// TwinCAT 3 PLC project BPC_PPA
// ProgramVersion: 3.1.4024.0
// libraries:
//   Tc2_Standard, * (Beckhoff Automation GmbH)
//   Tc2_System, * (Beckhoff Automation GmbH)
//   Tc3_Module, * (Beckhoff Automation GmbH)
//   VisuSymbols,3.5.10.0,System
// project tree:
//   / GlobalTextList.TcGTLO, PlcTask.TcTTO, Visualization Manager.TcVMO (not stored)
//   GVLs/ GVL.TcGVL, IO.TcGVL
//   POUs/ IOmap.TcPOU, MAIN.TcPOU, P_regulator.TcPOU
//   VISUs/ Visualization.TcVIS
// real-time tasks:
//   TASK PlcTask: cycle T#10ms, priority 20, ADS port 350

CONFIGURATION BPC_PPA
    RESOURCE PLC ON TwinCAT3
        TASK PlcTask(INTERVAL := T#10ms, PRIORITY := 20);
        PROGRAM MAIN WITH PlcTask : MAIN;
    END_RESOURCE
END_CONFIGURATION

// ---- GVLs/GVL.TcGVL
VAR_GLOBAL
    mb_Input_Coils : ARRAY [0..20] OF BOOL;
    mb_Output_Coils : ARRAY [0..20] OF BOOL;
    mb_Input_Registers : ARRAY [0..20] OF WORD;
    mb_Output_Registers : ARRAY [0..20] OF WORD;
END_VAR

// ---- GVLs/IO.TcGVL
{attribute 'qualified_only'}
VAR_GLOBAL
	// Analog Inputs
	StorageSupportPosition	: WORD;	// Pozice supportu skladovacího manipulátoru [0..27648]
	StorageCarriagePosition	: WORD;	// Pozice vozíku skladovacího manipulátoru [0..27648]
	
	// Digital Inputs
	SensorBoxStart			: BOOL;	// Sensor přítomnosti bedny na vstupu velkého dopravníkového pásu [0/1]
	SensorBoxHandling		: BOOL;	// Sensor přítomnosti bedny v pracovním prostoru překládacího manipulátoru [0/1]
	SensorBoxHandled		: BOOL;	// Sensor přítomnosti bedny na konci velkého dopravníkového pásu [0/1]
	SensorBoxStoring		: BOOL;	// Sensor přítomnosti bedny na naskladňovací pozici zakládacího dopravníku [0/1]
	SensorCanNew			: BOOL;	// Sensor přítomnosti nové plechovky na malém dopravníkovém pásu [0/1]
	SensorCanPrepare		: BOOL;	// Sensor přítomnosti plechovky uprostřed malého dopravníkového pásu [0/1]
	SensorCanHandling		: BOOL;	// Sensor přítomnosti plechovky v pracovním prostoru překládacího manipulátoru [0/1]
	ConvCanMoving			: BOOL;	// Signalizace pohybu motoru malého dopravníkového pásu [0/1]
	ConvBoxMoving			: BOOL;	// Signalizace pohybu motoru velkého dopravníkového pásu [0/1]
	ConvLoadMoving			: BOOL;	// Signalizace pohybu motoru zakládacího dopravníkového pásu [0/1]
	StorageSupportMoving	: BOOL;	// Signalizace pohybu motoru supportu skladovacího manipulátoru [0/1]
	StorageCarriageMoving	: BOOL;	// Signalizace pohybu motoru vozíku skladovacího manipulátoru [0/1]
	RoboticArmMoving		: BOOL;	// Signalizace vykonávání programového cyklu 6-osého robotického manipulátoru [0/1]
	HandlingMoving			: BOOL;	// Signalizace vykonávání programového cyklu překládacího manipulátoru [0/1]

	// Analog Outputs
	RoboticArmProgram		: WORD;	// Číslo programu pro vykonání 6-osým manipulátorem [0 .. základní pozice, 1 ..uchopení bedny, 2 .. položení bedny na pás]
	HandlingProgram			: WORD;	// Číslo programu pro vykonání překládacím manipulátorem [0 .. základní pozice, 1 .. přenesení na první pozici, 2 .. přenesení na druhou pozici, 3 .. přenesení na třetí pozici]
	ConvCanSpeed			: WORD;	// Rychlost motoru malého dopravníku [0..27648]
	ConvBoxSpeed			: WORD;	// Rychlost motoru velkého dopravníku [0..27648]
	ConvLoadSpeed			: WORD;	// Rychlost motoru zakládacího dopravníku [0..27648]
	StorageSupportSpeed		: WORD;	// Rychlost motoru supportu skladovacího manipulátoru [0..27648]
	StorageCarriageSpeed	: WORD;	// Rychlost motoru vozíku skladovacího manipulátoru [0..27648]
	
	// Digital Outputs
	RoboticArmStartCycle	: BOOL;	// Start programového cyklu 6-osého manipulátoru [náběžná hrana]
	HandlingStartCycle		: BOOL;	// Start programového cyklu překládacího manipulátoru [náběžná hrana]
	StorageLoad				: BOOL;	// Aktivace válce (ventilu) plošiny skladovacího manipulátoru DO naskladňovací polohy [0/1]
	StorageUnload			: BOOL;	// Aktivace válce (ventilu) plošiny skladovacího manipulátoru provyskladňovací polohy [0/1]
	ConvCanEnable			: BOOL;	// Povolení frekvenčního měniče motoru malého dopravníku [0/1]
	ConvCanForward			: BOOL;	// Aktivace chodu motoru malého dopravníku standardním směrem [0/1]
	ConvCanBackward			: BOOL;	// Aktivace chodu motoru malého dopravníku zpětným směrem [0/1]
	ConvBoxEnable			: BOOL;	// Povolení frekvenčního měniče motoru velkého dopravníku [0/1]
	ConvBoxForward			: BOOL;	// Aktivace chodu motoru velkého dopravníku standardním směrem [0/1]
	ConvBoxBackward			: BOOL;	// Aktivace chodu motoru velkého dopravníku zpětným směrem [0/1]
	ConvLoadEnable			: BOOL;	// Povolení frekvenčního měniče motoru zakládacího dopravníku [0/1]
	ConvLoadForward			: BOOL;	// Aktivace chodu motoru zakládacího dopravníku standardním směrem [0/1]
	ConvLoadBackward		: BOOL;	// Aktivace chodu motoru zakládacího dopravníku zpětným směrem [0/1]
	StorageSupportEnable	: BOOL;	// Povolení frekvenčního měniče motoru supportu skladovacího manipulátoru [0/1]
	StorageSupportForward	: BOOL;	// Aktivace chodu motoru supportu skladovacího manipulátoru standardním směrem [0/1]
	StorageSupportBackward	: BOOL;	// Aktivace chodu motoru supportu skladovacího manipulátoru zpětným směrem [0/1]
	StorageCarriageEnable	: BOOL;	// Povolení frekvenčního měniče motoru vozíku skladovacího manipuátoru [0/1]
	StorageCarriageForward	: BOOL;	// Aktivace chodu motoru vozíku skladovacího manipulátoru standardním směrem [0/1]
	StorageCarriageBackward	: BOOL;	// Aktivace chodu motoru vozíku skladovacího manipulátoru zpětným směrem [0/1]	
END_VAR

// ---- POUs/MAIN.TcPOU
PROGRAM MAIN
VAR CONSTANT
	//hlavni stavovy automat
	WAITING_FOR_START : USINT := 0;
	INIT_ROBOTS : USINT := 1; //inicializace handleru plechovek i velkeho robota
	INIT_ROBOTS_WAIT : USINT := 2; //cekaci stav, protoze pouzivam casovac
	GRAB_BOX : USINT := 3;
	GRAB_BOX_WAIT : USINT := 4;
	PUT_BOX : USINT := 5;
	PUT_BOX_WAIT : USINT := 6;
	DRIVE_BOX_TO_HANDLER : USINT := 7;
	HANDLE_CAN1 : USINT := 8;
	HANDLE_CAN1_WAIT : USINT := 9;
	HANDLE_CAN2 : USINT := 10;
	HANDLE_CAN2_WAIT : USINT := 11;
	HANDLE_CAN3 : USINT := 12;
	HANDLE_CAN3_WAIT : USINT := 13;
	CANS_HANDLED : USINT := 14;
	STORAGE_INIT : USINT := 15;
	STORAGE_INIT_WAIT : USINT := 16;
	GET_BOX_STORE : USINT := 17;
	GET_BOX_STORE_WAIT : USINT := 18;
	STORAGE_HANDLER_TO_BOX : USINT := 19;
	STORAGE_HANDLER_TO_BOX_WAIT: USINT := 20;
	LOAD_BOX : USINT := 21;
	LOAD_BOX_WAIT : USINT := 22;
	DRIVE_BOX_TO_STORE : USINT := 23;
	DRIVE_BOX_TO_STORE_WAIT : USINT := 24;
	BOX_UNLOAD : USINT := 25;
	BOX_UNLOAD_WAIT : USINT := 26;
	LAY_BOX : USINT := 27;
	STORING_DONE : USINT := 28;
END_VAR

VAR
	MainState : USINT := WAITING_FOR_START;
	StartProcess : BOOL := FALSE;
	CanSpeed : WORD := 1900;
	ConvSpeed : WORD := 2800;
	BoxAtTheEnd : BOOL := FALSE;
	TON_DelayCycle : TON;
	x : ARRAY [0..10] OF WORD := [25580, 23000, 20420, 17845, 15260, 12700, 10120, 7520, 4940, 2380, 750];
	y : ARRAY [0..5] OF WORD := [23750, 19142, 14535, 9927, 5318, 710];
	//FirstBoxDriven : BOOL := FALSE;
	BoxesStored : USINT := 0;
	ID : ARRAY [0..5] OF USINT := [2,5,6,3,9,4];
	P_RegulatorX : P_regulator;
	P_RegulatorY : P_regulator;
	yPosition : WORD := 0;
	xPosition : WORD := 0;
	RoboticArmStart : BOOL := FALSE;
	CentralStop : BOOL := FALSE;
END_VAR


IOmap(); //namapuj vstupy a vystupy
IF CentralStop THEN
	IO.ConvBoxEnable := 0;
	IO.ConvCanEnable := 0;
	IO.StorageSupportEnable := 0;
	IO.StorageCarriageEnable := 0;
	IO.StorageSupportEnable := 0;
END_IF

CASE MainState OF
	WAITING_FOR_START:
		IF StartProcess THEN
			MainState := INIT_ROBOTS;
		END_IF
		
	INIT_ROBOTS:
		IO.HandlingProgram := IO.RoboticArmProgram := 0;
		IO.HandlingStartCycle := IO.RoboticArmStartCycle := 1;
		TON_DelayCycle(IN := TRUE, PT := T#1S);
		IF TON_DelayCycle.Q THEN
			TON_DelayCycle(IN := 0);
			IF NOT IO.RoboticArmMoving AND NOT IO.HandlingMoving THEN
				IO.HandlingStartCycle := IO.RoboticArmStartCycle := 0;
				MainState := INIT_ROBOTS_WAIT;
			END_IF
		END_IF
		
	INIT_ROBOTS_WAIT:
		TON_DelayCycle(IN := TRUE, PT := T#1S);
		IF TON_DelayCycle.Q THEN
			TON_DelayCycle(IN := 0); 
			MainState := GRAB_BOX;
		END_IF
		
	GRAB_BOX:
		IO.RoboticArmProgram := 1;
		IO.RoboticArmStartCycle := 1;
		TON_DelayCycle(IN := TRUE, PT := T#1S);
		IF TON_DelayCycle.Q THEN
			TON_DelayCycle(IN := 0);
			IF NOT IO.RoboticArmMoving THEN
				IO.RoboticArmStartCycle := 0;
				MainState := GRAB_BOX_WAIT;
			END_IF
		END_IF
		
	GRAB_BOX_WAIT:
		TON_DelayCycle(IN := TRUE, PT := T#1S);
		IF TON_DelayCycle.Q THEN
			TON_DelayCycle(IN := 0);
			MainState := PUT_BOX;
		END_IF
	
	PUT_BOX:
		IO.RoboticArmProgram := 2;
		IO.RoboticArmStartCycle := 1;
		TON_DelayCycle(IN := TRUE, PT := T#1S);
		IF TON_DelayCycle.Q THEN 
			TON_DelayCycle(IN := 0);
			IF NOT IO.RoboticArmMoving THEN
				IO.RoboticArmStartCycle := 0;
				MainState := PUT_BOX_WAIT;
			END_IF
			
		END_IF
		
	PUT_BOX_WAIT:
		TON_DelayCycle(IN := TRUE, PT := T#1S);
		IF TON_DelayCycle.Q THEN
			TON_DelayCycle(IN := 0);
			MainState := DRIVE_BOX_TO_HANDLER;
		END_IF
		
	DRIVE_BOX_TO_HANDLER:
		
		IF IO.SensorBoxHandling THEN
			IO.ConvBoxEnable := 0;
			MainState := HANDLE_CAN1;
		ELSE
			IO.ConvBoxEnable := 1;
		END_IF
		
		
	HANDLE_CAN1:
		IO.HandlingProgram := 1;
		IO.HandlingStartCycle := 1;
		TON_DelayCycle(IN := TRUE, PT := T#1S);
		IF TON_DelayCycle.Q THEN
			TON_DelayCycle(IN := 0);
			IF NOT IO.HandlingMoving THEN
				IO.HandlingStartCycle := 0; 
				MainState := HANDLE_CAN1_WAIT;
			END_IF
		END_IF
		
	HANDLE_CAN1_WAIT:
		TON_DelayCycle(IN := TRUE, PT := T#1S);
		IF TON_DelayCycle.Q THEN
			TON_DelayCycle(IN := 0); 
			MainState := HANDLE_CAN2;
		END_IF
		
	HANDLE_CAN2:
		TON_DelayCycle(IN := TRUE, PT := T#1S);
		IO.HandlingProgram := 2;
		IO.HandlingStartCycle := 1;
		IF TON_DelayCycle.Q THEN
			TON_DelayCycle(IN := 0);
			IF NOT IO.HandlingMoving THEN
				IO.HandlingStartCycle := 0;
				MainState := HANDLE_CAN2_WAIT;
			END_IF
		END_IF
		
	HANDLE_CAN2_WAIT:
		TON_DelayCycle(IN := TRUE, PT := T#1S);
		IF TON_DelayCycle.Q THEN
			TON_DelayCycle(IN := 0); 
			MainState := HANDLE_CAN3;
		END_IF
		
	HANDLE_CAN3:
		TON_DelayCycle(IN := TRUE, PT := T#1S);
		IO.HandlingProgram := 3;
		IO.HandlingStartCycle := 1;
		IF TON_DelayCycle.Q THEN
			TON_DelayCycle(IN := 0);
			IF NOT IO.HandlingMoving THEN
				IO.HandlingStartCycle := 0; 
				MainState := HANDLE_CAN3_WAIT;
			END_IF
		END_IF
		
	HANDLE_CAN3_WAIT:
		TON_DelayCycle(IN := TRUE, PT := T#1S);
		IF TON_DelayCycle.Q THEN
			TON_DelayCycle(IN := 0);
			MainState := CANS_HANDLED;
		END_IF	
	
	CANS_HANDLED:
		MainState := GET_BOX_STORE;
		IO.ConvBoxEnable := 1;
	
	STORAGE_INIT:
		TON_DelayCycle(IN := TRUE, PT := T#1S);
		
		P_RegulatorX.SetpointPos := 750;
		P_RegulatorY.SetpointPos := 1100;
		
		IF TON_DelayCycle.Q THEN
			TON_DelayCycle(IN := 0);
			IF NOT IO.StorageCarriageMoving AND NOT IO.StorageSupportMoving THEN
				
				MainState := STORAGE_INIT_WAIT;
			END_IF
		
		END_IF
		
	STORAGE_INIT_WAIT:
		TON_DelayCycle(IN := TRUE, PT := T#1S);
		IF TON_DelayCycle.Q THEN
			TON_DelayCycle(IN := 0); 
			MainState := GET_BOX_STORE;
		END_IF
		
	GET_BOX_STORE:
		IO.StorageCarriageEnable := IO.StorageSupportEnable := 1;
		IF IO.SensorBoxStoring THEN
			TON_DelayCycle(IN := TRUE, PT := T#1S);
			P_RegulatorX.SetpointPos := 750;
			P_RegulatorY.SetpointPos := 1100;	
			IF TON_DelayCycle.Q THEN
					IF NOT IO.StorageSupportMoving AND NOT IO.StorageCarriageMoving THEN
						
						MainState := GET_BOX_STORE_WAIT;
					END_IF
			END_IF
		END_IF
		
	GET_BOX_STORE_WAIT:
		TON_DelayCycle(IN := TRUE, PT := T#1S);
		IF TON_DelayCycle.Q THEN
			TON_DelayCycle(IN := 0); 
			
			MainState := STORAGE_HANDLER_TO_BOX;
		END_IF
		
	STORAGE_HANDLER_TO_BOX:
		TON_DelayCycle(IN := TRUE, PT := T#2S);
		IF TON_DelayCycle.Q THEN
			P_RegulatorY.SetpointPos := 2100;
			IO.StorageLoad := 1;
			MainState := STORAGE_HANDLER_TO_BOX_WAIT;
		END_IF
	
	STORAGE_HANDLER_TO_BOX_WAIT:
		TON_DelayCycle(IN := TRUE, PT := T#2S);
		IF TON_DelayCycle.Q THEN
			
			TON_DelayCycle(IN := FALSE);
			MainState := LOAD_BOX;
		END_IF
		
	LOAD_BOX:
		TON_DelayCycle(IN := TRUE, PT := T#2S);
		IF TON_DelayCycle.Q THEN
			TON_DelayCycle(IN := FALSE);
			IO.StorageLoad := 0;
			MainState := LOAD_BOX_WAIT;
		END_IF
		
	LOAD_BOX_WAIT:
		TON_DelayCycle(IN := TRUE, PT := T#2S);
		IF TON_DelayCycle.Q THEN
			TON_DelayCycle(IN := FALSE);
			MainState := DRIVE_BOX_TO_STORE;
		END_IF
	
		
	DRIVE_BOX_TO_STORE: 
		TON_DelayCycle(IN := TRUE, PT := T#1S);
		IF TON_DelayCycle.Q THEN
			TON_DelayCycle(IN := FALSE);
				P_RegulatorX.SetpointPos := x[ID[BoxesStored]];
				P_RegulatorY.SetpointPos := y[BoxesStored] + 400;
			MainState := DRIVE_BOX_TO_STORE_WAIT; 
		END_IF
		
	DRIVE_BOX_TO_STORE_WAIT:
		TON_DelayCycle(IN := TRUE, PT := T#1S);
		IF TON_DelayCycle.Q THEN
			TON_DelayCycle(IN := FALSE);
			MainState := BOX_UNLOAD;
		END_IF
		
	BOX_UNLOAD: 
		TON_DelayCycle(IN := TRUE, PT := T#1S);
		IF TON_DelayCycle.Q THEN
			IF NOT IO.StorageCarriageMoving AND NOT IO.StorageSupportMoving THEN
				TON_DelayCycle(IN := FALSE);
				IO.StorageUnload := 1;
				MainState := BOX_UNLOAD_WAIT;
			END_IF
		END_IF
	BOX_UNLOAD_WAIT:
		TON_DelayCycle(IN := TRUE, PT := T#1S);
		IF TON_DelayCycle.Q THEN
				TON_DelayCycle(IN := FALSE);
				MainState := LAY_BOX;
				P_RegulatorY.SetpointPos := P_RegulatorY.SetpointPos - 400;
		END_IF
		
	LAY_BOX:
		TON_DelayCycle(IN := TRUE, PT := T#1S);
		IF TON_DelayCycle.Q THEN
			IF NOT IO.StorageCarriageMoving AND NOT IO.StorageSupportMoving THEN
				TON_DelayCycle(IN := FALSE);
				IO.StorageUnload := 0;
				IF BoxesStored < 5 THEN
					MainState := GRAB_BOX;
					BoxesStored := BoxesStored + 1;
				ELSE
					MainState := STORING_DONE;
				END_IF
			END_IF 
			
		END_IF
		
END_CASE

IF IO.SensorBoxHandled THEN
	BoxAtTheEnd := TRUE;
END_IF

//maly dopravnik
IO.ConvCanSpeed := CanSpeed;
IO.ConvCanForward := TRUE;
IO.ConvCanEnable := NOT IO.SensorCanHandling AND MainState > WAITING_FOR_START;
StartProcess := FALSE;

//velky dopravnik
IO.ConvBoxSpeed := ConvSpeed;
IO.ConvBoxForward := TRUE;

//zakladaci dopravnik
IO.ConvLoadSpeed := ConvSpeed;
IO.ConvLoadForward := TRUE;
IO.ConvLoadEnable := BoxAtTheEnd AND NOT IO.SensorBoxStoring;

P_RegulatorX(CurrentPos := IO.StorageSupportPosition, DecelerationLength := 15000);
IO.StorageSupportSpeed := REAL_TO_WORD(P_RegulatorX.Speed);
IO.StorageSupportForward := P_RegulatorX.MoveForward;
IO.StorageSupportBackward := P_RegulatorX.MoveBackward;

P_RegulatorY(CurrentPos := IO.StorageCarriagePosition, DecelerationLength := 17000);
IO.StorageCarriageSpeed := REAL_TO_WORD(P_RegulatorY.Speed);
IO.StorageCarriageForward := P_RegulatorY.MoveForward;
IO.StorageCarriageBackward := P_RegulatorY.MoveBackward;

END_PROGRAM

// ---- POUs/P_regulator.TcPOU
FUNCTION_BLOCK P_regulator
VAR CONSTANT
    //FSM states
    NOT_MOVING : USINT := 0;
    MOVING : USINT := 1;

    OUTER_POS_TOL : REAL := 10;
    INNER_POS_TOL : REAL := 5;

END_VAR

VAR
    MoveState : USINT := NOT_MOVING;

    DesiredSpeed : REAL;
    DecelerationRatio : REAL;

END_VAR

VAR_INPUT
    CurrentPos : REAL;
    SetpointPos : REAL;
    MaxSpeed : REAL := 13000;
    DecelerationLength : REAL := 18000;
END_VAR

VAR_OUTPUT
    Speed : REAL;
    MoveForward : BOOL;
    MoveBackward : BOOL;
END_VAR

CASE MoveState OF
    NOT_MOVING:
        IF SetpointPos - CurrentPos > OUTER_POS_TOL THEN
            MoveForward := TRUE;
            MoveBackward := FALSE;
            MoveState := MOVING;
        ELSIF CurrentPos - SetpointPos > OUTER_POS_TOL THEN
            MoveForward := FALSE;
            MoveBackward := TRUE;
            MoveState := MOVING;
        END_IF

    MOVING:
        IF NOT (MoveForward AND SetpointPos - CurrentPos < INNER_POS_TOL OR MoveBackward AND CurrentPos - SetpointPos < INNER_POS_TOL) THEN
           IF DecelerationLength > 0 THEN
				DecelerationRatio := ABS(SetpointPos - CurrentPos) / DecelerationLength;
				IF DecelerationRatio > 1 THEN
					DecelerationRatio := 1;
				END_IF
			ELSE
				DecelerationRatio := 1;
			END_IF
            DesiredSpeed := MaxSpeed * DecelerationRatio;
        ELSE
			DesiredSpeed := 0;
            MoveForward := MoveBackward := FALSE;
            MoveState := NOT_MOVING;
			
        END_IF

END_CASE
Speed := DesiredSpeed;

END_FUNCTION_BLOCK

// ---- POUs/IOmap.TcPOU
PROGRAM IOmap
VAR
END_VAR

// Analog Inputs
IO.StorageSupportPosition 		:= GVL.mb_Output_Registers[1];		// Pozice supportu skladovacího manipulátoru [0..27648]
IO.StorageCarriagePosition 		:= GVL.mb_Output_Registers[2];		// Pozice vozíku skladovacího manipulátoru [0..27648]
	
// Digital Inputs
IO.SensorBoxStart 				:= GVL.mb_Output_Registers[0].0;	// Sensor přítomnosti bedny na vstupu velkého dopravníkového pásu [0/1]
IO.SensorBoxHandling 			:= GVL.mb_Output_Registers[0].1;	// Sensor přítomnosti bedny v pracovním prostoru překládacího manipulátoru [0/1]
IO.SensorBoxHandled 			:= GVL.mb_Output_Registers[0].2;	// Sensor přítomnosti bedny na konci velkého dopravníkového pásu [0/1]
IO.SensorBoxStoring 			:= GVL.mb_Output_Registers[0].3;	// Sensor přítomnosti bedny na naskladňovací pozici zakládacího dopravníku [0/1]
IO.SensorCanNew 				:= GVL.mb_Output_Registers[0].4;	// Sensor přítomnosti nové plechovky na malém dopravníkovém pásu [0/1]
IO.SensorCanPrepare 			:= GVL.mb_Output_Registers[0].5;	// Sensor přítomnosti plechovky uprostřed malého dopravníkového pásu [0/1]
IO.SensorCanHandling 			:= GVL.mb_Output_Registers[0].6;	// Sensor přítomnosti plechovky v pracovním prostoru překládacího manipulátoru [0/1]
IO.ConvCanMoving 				:= GVL.mb_Output_Registers[0].7;	// Signalizace pohybu motoru malého dopravníkového pásu [0/1]
IO.ConvBoxMoving 				:= GVL.mb_Output_Registers[0].8;	// Signalizace pohybu motoru velkého dopravníkového pásu [0/1]
IO.ConvLoadMoving 				:= GVL.mb_Output_Registers[0].9;	// Signalizace pohybu motoru zakládacího dopravníkového pásu [0/1]
IO.StorageSupportMoving 		:= GVL.mb_Output_Registers[0].10;	// Signalizace pohybu motoru supportu skladovacího manipulátoru [0/1]
IO.StorageCarriageMoving 		:= GVL.mb_Output_Registers[0].11;	// Signalizace pohybu motoru vozíku skladovacího manipulátoru [0/1]
IO.RoboticArmMoving 			:= GVL.mb_Output_Registers[0].12;	// Signalizace vykonávání programového cyklu 6-osého robotického manipulátoru [0/1]
IO.HandlingMoving 				:= GVL.mb_Output_Registers[0].13;	// Signalizace vykonávání programového cyklu překládacího manipulátoru [0/1]

// Analog Outputs
GVL.mb_Input_Registers[2] 		:= IO.RoboticArmProgram;			// Číslo programu pro vykonání 6-osým manipulátorem [0 .. základní pozice, 1 ..uchopení bedny, 2 .. položení bedny na pás]
GVL.mb_Input_Registers[3] 		:= IO.HandlingProgram;				// Číslo programu pro vykonání překládacím manipulátorem [0 .. základní pozice, 1 .. přenesení na první pozici, 2 .. přenesení na druhou pozici, 3 .. přenesení na třetí pozici]
GVL.mb_Input_Registers[4] 		:= IO.ConvCanSpeed;					// Rychlost motoru malého dopravníku [0..27648]
GVL.mb_Input_Registers[5] 		:= IO.ConvBoxSpeed;					// Rychlost motoru velkého dopravníku [0..27648]
GVL.mb_Input_Registers[6] 		:= IO.ConvLoadSpeed;				// Rychlost motoru zakládacího dopravníku [0..27648]
GVL.mb_Input_Registers[7] 		:= IO.StorageSupportSpeed;			// Rychlost motoru supportu skladovacího manipulátoru [0..27648]
GVL.mb_Input_Registers[8] 		:= IO.StorageCarriageSpeed;			// Rychlost motoru vozíku skladovacího manipulátoru [0..27648]

// Digital Outputs
GVL.mb_Input_Registers[0].0 	:= IO.RoboticArmStartCycle;			// Start programového cyklu 6-osého manipulátoru [náběžná hrana]
GVL.mb_Input_Registers[0].1 	:= IO.HandlingStartCycle;			// Start programového cyklu překládacího manipulátoru [náběžná hrana]
GVL.mb_Input_Registers[0].2 	:= IO.StorageLoad;					// Aktivace válce (ventilu) plošiny skladovacího manipulátoru DO naskladňovací polohy [0/1]
GVL.mb_Input_Registers[0].3 	:= IO.StorageUnload;				// Aktivace válce (ventilu) plošiny skladovacího manipulátoru provyskladňovací polohy [0/1]
GVL.mb_Input_Registers[0].4 	:= IO.ConvCanEnable;				// Povolení frekvenčního měniče motoru malého dopravníku [0/1]
GVL.mb_Input_Registers[0].5 	:= IO.ConvCanForward;				// Aktivace chodu motoru malého dopravníku standardním směrem [0/1]
GVL.mb_Input_Registers[0].6 	:= IO.ConvCanBackward;				// Aktivace chodu motoru malého dopravníku zpětným směrem [0/1]
GVL.mb_Input_Registers[0].7 	:= IO.ConvBoxEnable;				// Povolení frekvenčního měniče motoru velkého dopravníku [0/1]
GVL.mb_Input_Registers[0].8 	:= IO.ConvBoxForward;				// Aktivace chodu motoru velkého dopravníku standardním směrem [0/1]
GVL.mb_Input_Registers[0].9 	:= IO.ConvBoxBackward;				// Aktivace chodu motoru velkého dopravníku zpětným směrem [0/1]
GVL.mb_Input_Registers[0].10 	:= IO.ConvLoadEnable;				// Povolení frekvenčního měniče motoru zakládacího dopravníku [0/1]
GVL.mb_Input_Registers[0].11 	:= IO.ConvLoadForward;				// Aktivace chodu motoru zakládacího dopravníku standardním směrem [0/1]
GVL.mb_Input_Registers[0].12 	:= IO.ConvLoadBackward;				// Aktivace chodu motoru zakládacího dopravníku zpětným směrem [0/1]
GVL.mb_Input_Registers[0].13 	:= IO.StorageSupportEnable;			// Povolení frekvenčního měniče motoru supportu skladovacího manipulátoru [0/1]
GVL.mb_Input_Registers[0].14 	:= IO.StorageSupportForward;		// Aktivace chodu motoru supportu skladovacího manipulátoru standardním směrem [0/1]
GVL.mb_Input_Registers[0].15 	:= IO.StorageSupportBackward;		// Aktivace chodu motoru supportu skladovacího manipulátoru zpětným směrem [0/1]
GVL.mb_Input_Registers[1].0 	:= IO.StorageCarriageEnable;		// Povolení frekvenčního měniče motoru vozíku skladovacího manipuátoru [0/1]
GVL.mb_Input_Registers[1].1 	:= IO.StorageCarriageForward;		// Aktivace chodu motoru vozíku skladovacího manipulátoru standardním směrem [0/1]
GVL.mb_Input_Registers[1].2 	:= IO.StorageCarriageBackward;		// Aktivace chodu motoru vozíku skladovacího manipulátoru zpětným směrem [0/1]

END_PROGRAM

// ---- GlobalTextList.TcGTLO
TEXTLIST GlobalTextList
  32 = '6osý manipulátor'
  732 = 'Bedna na konci skladovacího dopravníku'
  722 = 'Bedna na konci skladovacího pásu'
  892 = 'Bedna na konci velkého pásového dopravníku'
  391 = 'Bedna na konci velkého pásu'
  393 = 'Bedna na začátku velkého pásového dopravníku'
  428 = 'Bedna na začátku velkého pásu'
  990 = 'Bedna v nakládacím prostoru plechovek'
  873 = 'GroupBox'
  315 = 'Hlavní vypínač'
  939 = 'Hýbe se'
  377 = 'Konec velkého pásu'
  67 = 'Lalal'
  290 = 'Lalalal'
  544 = 'Manipulátor plechovek'
  502 = 'Plechovka na konci pásu plechovek'
  364 = 'Plechovka na konci velkého pásu'
  329 = 'Plechovka na začátku dopravníku plechovek'
  462 = 'Plechovka na začátku velkého pásu'
  573 = 'Plechovka v nakládacím prostoru do krabice'
  188 = 'Senzory'
  89 = 'Senzory bedny'
  458 = 'Senzory plechovky'
  942 = 'Start'
  635 = 'Start velkého pásu'
END_TEXTLIST

// ---- VISUs/Visualization.TcVIS
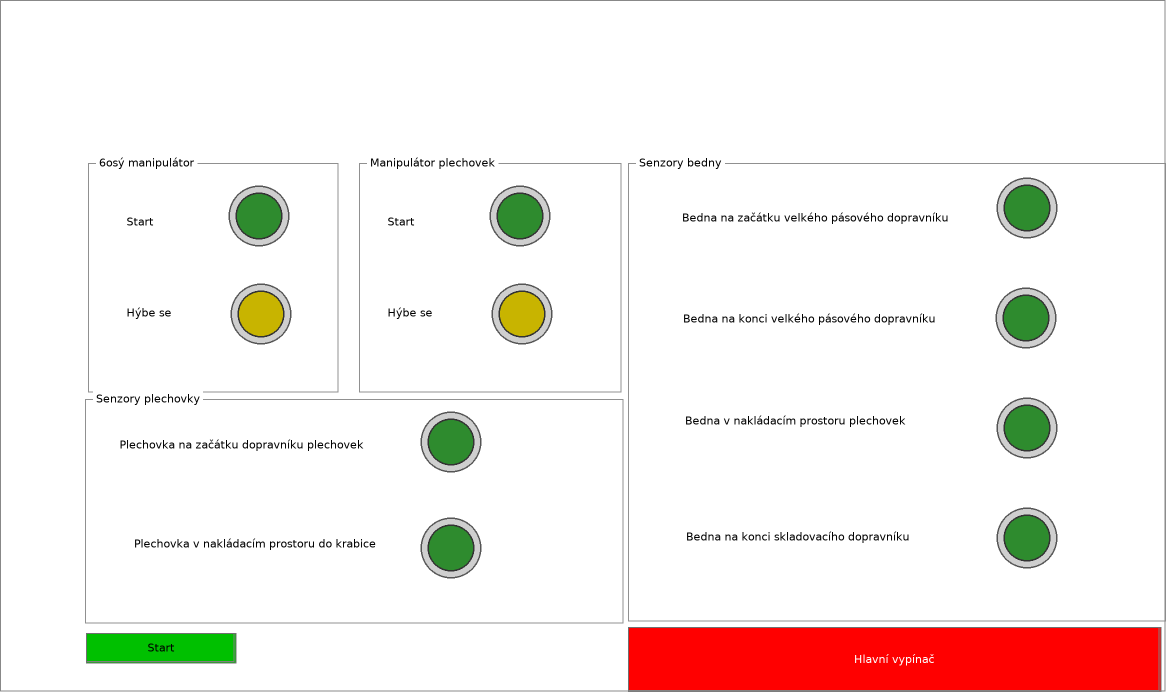
VISUALIZATION Visualization  // 1166x692
    Lamp1 (992,173 70x70), variable: IO.SensorBoxStart, style: Lamp-Lamp1-Green
    Lamp1 (991,283 70x70), variable: IO.SensorBoxHandled, style: Lamp-Lamp1-Green
    Label (669,203 293x30), "Bedna na začátku velkého pásového dopravníku"
    Label (663,304 293x30), "Bedna na konci velkého pásového dopravníku"
    Lamp1 (992,393 70x70), variable: IO.SensorBoxHandling, style: Lamp-Lamp1-Green
    Label (644,406 303x30), "Bedna v nakládacím prostoru plechovek"
    Lamp1 (992,503 70x70), variable: IO.SensorBoxStoring, style: Lamp-Lamp1-Green
    Label (668,522 260x30), "Bedna na konci skladovacího dopravníku"
    GroupBox (628,155 538x466), "Senzory bedny"
    Lamp1 (485,181 70x70), variable: IO.HandlingStartCycle, style: Lamp-Lamp1-Green
    Label (356,301 108x24), "Hýbe se"
    Lamp1 (487,279 70x70), variable: IO.HandlingMoving, style: Lamp-Lamp1-Yellow
    Label (347,208 108x28), "Start"
    Lamp1 (224,181 70x70), variable: IO.RoboticArmStartCycle, style: Lamp-Lamp1-Green
    Label (95,301 108x24), "Hýbe se"
    Lamp1 (226,279 70x70), variable: IO.RoboticArmMoving, style: Lamp-Lamp1-Yellow
    Label (86,208 108x28), "Start"
    GroupBox (88,155 250x237), "6osý manipulátor"
    GroupBox (359,155 262x237), "Manipulátor plechovek"
    Button (628,627 533x65), "Hlavní vypínač", invisible if: MAIN.StartProcess
        toggle MAIN.CentralStop
    Button (86,633 150x30), "Start"
        toggle MAIN.StartProcess
    Lamp1 (416,407 70x70), variable: IO.SensorCanNew, style: Lamp-Lamp1-Green
    Label (114,430 255x30), "Plechovka na začátku dopravníku plechovek"
    Lamp1 (416,513 70x70), variable: IO.SensorCanHandling, style: Lamp-Lamp1-Green
    GroupBox (85,391 538x232), "Senzory plechovky"
    Label (118,529 274x30), "Plechovka v nakládacím prostoru do krabice"
END_VISUALIZATION
